TYPE (* logiBUS 2 CAN DI Struct Octal *)
  (* Version 1.0, 2026-05-28, franz *)
  PACKAGE logiBUS::io::DI_CAN;
  logiBUS_2_CAN_DI_S_Octal : STRUCT
    Port1 : logiBUS::io::DI_CAN::logiBUS_2_CAN_DI_S := (Pin := 255);
    Port2 : logiBUS::io::DI_CAN::logiBUS_2_CAN_DI_S := (Pin := 255);
    Port3 : logiBUS::io::DI_CAN::logiBUS_2_CAN_DI_S := (Pin := 255);
    Port4 : logiBUS::io::DI_CAN::logiBUS_2_CAN_DI_S := (Pin := 255);
    Port5 : logiBUS::io::DI_CAN::logiBUS_2_CAN_DI_S := (Pin := 255);
    Port6 : logiBUS::io::DI_CAN::logiBUS_2_CAN_DI_S := (Pin := 255);
    Port7 : logiBUS::io::DI_CAN::logiBUS_2_CAN_DI_S := (Pin := 255);
    Port8 : logiBUS::io::DI_CAN::logiBUS_2_CAN_DI_S := (Pin := 255);
  END_STRUCT;
END_TYPE
